Staubli VAL3: onF6Event.pgx

program onF6Event(string x_sName)
begin
  // look if the bButton is enable
  if bButton[5]
    // RESET
    call pallet:setPalletPos(x_sName,0)
    // refresh it
    call buildList()
    use:bUseRefresh=true
  endIf
end
